FUNCTION_BLOCK UnitTestOnlyMatchingNames EXTENDS FB_TestSuite

METHOD HasMatchingName
TEST('HasMatchingName');

AssertTrue(Condition:=TRUE, Message:='Blabla');

TEST_FINISHED();
END_METHOD

METHOD NameAlsoMatches
VAR_INPUT
END_VAR
TEST('NameAlsoMatches');

AssertTrue(Condition:=TRUE, Message:='Blabla');

TEST_FINISHED();
END_METHOD

END_FUNCTION_BLOCK

(* stored: Version 1.1.0.1, ProductVersion 3.1.4024.12
   POU UnitTestOnlyMatchingNames: Id {bfb9981c-9c74-4219-8ca5-1996ef8ad405}, SpecialFunc None
   Method HasMatchingName: Id {1e1b8b4b-4792-4ed6-8da9-fd826de17784}
   Method NameAlsoMatches: Id {21882d82-3823-4341-a489-b0fbf5d5c4eb} *)
